PROGRAM pouDataDisplay
VAR
	werd: DWORD;
	dataCombi: ARRAY[0..15] OF FB_DataCombine;
	i: INT;
	
END_VAR

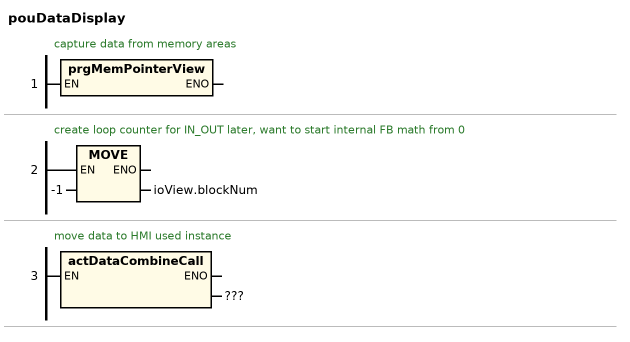
// NETWORK 1
// capture data from memory areas
prgMemPointerView();

// NETWORK 2
// create loop counter for IN_OUT later, want to start internal FB math from 0
ioView.blockNum := -1;

// NETWORK 3
// move data to HMI used instance
actDataCombineCall();

ACTION actDataCombineCall:
//call data for each row
FOR i:=0 TO 15 DO
	
	datacombi[i](iWordData:=ioView.ViewingArray[i],
				 iRealHEXConv:=ioView.memHexDisplay,
				 iWordSize:= ioView.memsize,
				 blockCount:= ioView.blockNum);

	ioView.ByteRow[i]:=dataCombi[i].outputRow;
	

END_FOR
END_ACTION

END_PROGRAM

(* stored: Version 1.1.0.1, ProductVersion 3.1.4024.12
   POU pouDataDisplay: Id {9d244046-dbb0-4950-8033-df6cea4a2323}, SpecialFunc None
   Action actDataCombineCall: Id {5fb03654-dc97-4cb1-987a-81f27fdba4f1} *)
